FUNCTION_BLOCK FB_Klep IMPLEMENTS ITF_UnitKlep
VAR
    _cmdOpen : BOOL;   // command naar de klep
    _isOpen  : BOOL;   // status van de klep
END_VAR

_isOpen := _cmdOpen; // Simpele logica: status volgt command

PROPERTY PUBLIC CmdOpen : BOOL
GET
CmdOpen := _cmdOpen;     // uitlezen command
END_GET
SET
_cmdOpen := CmdOpen;     // schrijven naar command
END_SET
END_PROPERTY

PROPERTY PUBLIC IsOpen : BOOL
GET
IsOpen := _isOpen;   // status van de klep
END_GET
SET
END_SET
END_PROPERTY

END_FUNCTION_BLOCK

(* stored: Version 1.1.0.1
   POU FB_Klep: Id {a42b2b1d-3d0d-4ad8-8a49-e659df0386f5}, SpecialFunc None
   Property CmdOpen: Id {86f25ea2-b0fc-4cd7-bc06-affc0226726a}
   Get Get: Id {92e1e3a2-8e91-40b3-819a-04f0a5ac7e56}
   Set Set: Id {b3f01c57-32cd-4802-9c11-07a62a96f994}
   Property IsOpen: Id {31527c57-edc2-4678-9abe-6ccf7774afd3}
   Get Get: Id {a536c20e-7137-476a-a29c-e85d6f2b2297}
   Set Set: Id {8ca1fbf7-f843-4dc9-ae5c-1c69c5f94f11} *)
